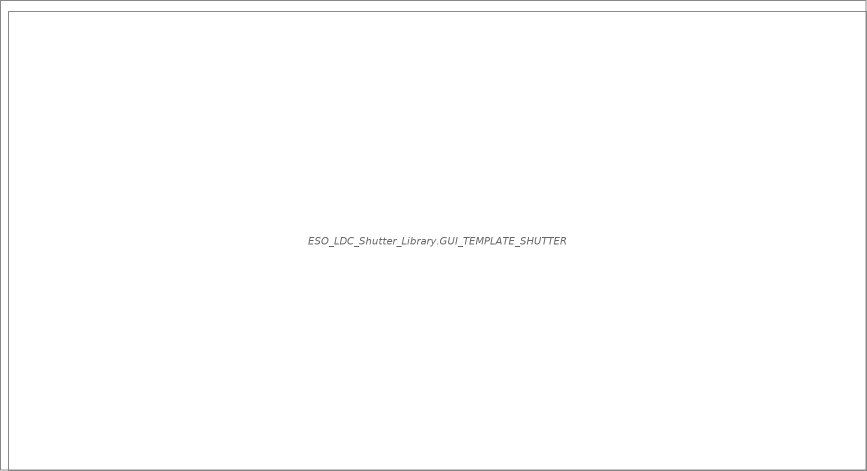
VISUALIZATION Shutter_1  // 867x471
    Frame (8,11 859x460)
        shows ESO_LDC_Shutter_Library.GUI_TEMPLATE_SHUTTER(m_Instance := MAIN.shutter_1)
END_VISUALIZATION

(* stored: Version 1.1.0.1, ProductVersion 3.1.4024.12
   Visu Shutter_1: Id {2c82cc8c-95ba-41cf-9646-7cc08c256d31} *)
